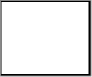
VISUALIZATION VISU_SystemButton  // 92x77
VAR_IN_OUT
    widget : SystemButtonWidget;
END_VAR
    Rectangle (0,0 90x75), invisible if: widget.isNotOrange
    Rectangle (0,0 90x75), invisible if: widget.isNotGray
    Rectangle (0,0 90x75), invisible if: widget.isNotBlue
    Rectangle (0,0 90x75), invisible if: widget.isNotRed
    Rectangle (0,0 90x75), invisible if: widget.isNotGreen
    Rectangle (0,50 90x25), "%s", text variable: widget.name
    Image (25,10 40x40), image: VISU_SystemButtonImages.Home
        p84334746: widget.name
    Rectangle (0,0 90x75), invisible if: widget.notActivated
    Line (0,74) (90,74), invisible if: widget.activated
    Line (89,75) (89,0), invisible if: widget.activated
    Line (0,74) (0,0), invisible if: widget.activated
    Line (88,0) (0,0), invisible if: widget.activated
    Line (0,1) (90,1), invisible if: widget.notActivated
    Line (1,75) (1,0), invisible if: widget.notActivated
    Line (90,75) (1,75), invisible if: widget.notActivated
    Line (90,75) (90,1), invisible if: widget.notActivated
END_VISUALIZATION

(* stored: Version 1.1.0.1, ProductVersion 3.1.4019.2
   Visu VISU_SystemButton: Id {0954f149-abc0-40b6-bcbc-693b1b9eaed9} *)
